(* IEC 61131-3 sources: RL_MAR/experiments/comparison/llm4plc/results/gpt-4o-mini_20260506_100619/20260506_102027, 2 files *)

(* ---- generated_code_iteration_0.st ---- *)
ructured-text
START_ST
FUNCTION_BLOCK WindTurbineControl
VAR_INPUT
    WindSpeedSensor : REAL; (* Input for measuring wind speed *)
    GeneratorSpeedSensor : REAL; (* Input for measuring generator speed *)
END_VAR

VAR_OUTPUT
    BladePitch : INT; (* Output for blade pitch control (degrees) *)
    GeneratorSpeed : REAL; (* Output for generator speed control (RPM) *)
END_VAR

VAR
    state : INT; (* The state variable to track current state *)
    prevState : INT; (* The previous state variable (optional for state change logic) *)
    WindSpeed : REAL; (* The current wind speed from WindSpeedSensor *)
    GeneratorSpeed : REAL; (* The current generator speed from GeneratorSpeedSensor *)
END_VAR

(* Initialize the state variable to a default state (LOW WIND SPEED) *)
state := 0;

(* Main control logic *)
IF WindSpeedSensor <= 3.0 THEN
    state := 0; (* LOW WIND SPEED *)
ELSIF WindSpeedSensor > 3.0 AND WindSpeedSensor <= 5.0 THEN
    state := 1; (* MODERATE WIND SPEED *)
ELSIF WindSpeedSensor > 5.0 THEN
    state := 2; (* HIGH WIND SPEED *)
END_IF;

(* Set outputs based on the current state *)
CASE state OF
    0: (* LOW WIND SPEED *)
        BladePitch := -5;
        GeneratorSpeed := 500;
    1: (* MODERATE WIND SPEED *)
        BladePitch := 0;
        GeneratorSpeed := 800;
    2: (* HIGH WIND SPEED *)
        BladePitch := 5;
        GeneratorSpeed := 1000;
END_CASE;

END_FUNCTION_BLOCK
END_ST

(* ---- generated_code_iteration_1.st ---- *)
START_REASON
The errors in the original Structured Text (ST) code occurred due to the declaration of the variable `GeneratorSpeed` in both the VAR_OUTPUT and VAR sections. This resulted in a naming conflict, as the same variable name cannot be used for both output and local variable declarations within the same function block. To resolve this issue, I will rename the local variable to avoid the conflict and ensure the code adheres to the required structure.
END_REASON

START_ST
FUNCTION_BLOCK WindTurbineControl
VAR_INPUT
    WindSpeedSensor : REAL; (* Input for measuring wind speed *)
    GeneratorSpeedSensor : REAL; (* Input for measuring generator speed *)
END_VAR

VAR_OUTPUT
    BladePitch : INT; (* Output for blade pitch control (degrees) *)
    GeneratorSpeed : REAL; (* Output for generator speed control (RPM) *)
END_VAR

VAR
    state : INT; (* The state variable to track current state *)
    prevState : INT; (* The previous state variable (optional for state change logic) *)
    WindSpeed : REAL; (* The current wind speed from WindSpeedSensor *)
    CurrentGeneratorSpeed : REAL; (* Renamed local variable to avoid conflict *)
END_VAR

(* Initialize the state variable to a default state (LOW WIND SPEED) *)
state := 0;

(* Main control logic *)
IF WindSpeedSensor <= 3.0 THEN
    state := 0; (* LOW WIND SPEED *)
ELSIF WindSpeedSensor > 3.0 AND WindSpeedSensor <= 5.0 THEN
    state := 1; (* MODERATE WIND SPEED *)
ELSIF WindSpeedSensor > 5.0 THEN
    state := 2; (* HIGH WIND SPEED *)
END_IF;

(* Set outputs based on the current state *)
CASE state OF
    0: (* LOW WIND SPEED *)
        BladePitch := -5;
        CurrentGeneratorSpeed := 500;
    1: (* MODERATE WIND SPEED *)
        BladePitch := 0;
        CurrentGeneratorSpeed := 800;
    2: (* HIGH WIND SPEED *)
        BladePitch := 5;
        CurrentGeneratorSpeed := 1000;
END_CASE;

(* Assign the local generator speed to the output variable *)
GeneratorSpeed := CurrentGeneratorSpeed;

END_FUNCTION_BLOCK
END_ST
